INTERFACE I_Axis

METHOD PrepareDecoupling : I_Axis
VAR_INPUT
	slaveAxis : REFERENCE TO AXIS_REF;
	slaveStatus : REFERENCE TO ST_AXISSTATUS;
END_VAR
END_METHOD

METHOD StartCoupling : I_Axis
VAR_INPUT
END_VAR
END_METHOD

METHOD StartDecoupling : BOOL
VAR_INPUT
END_VAR
END_METHOD

METHOD StartHoming : BOOL;
VAR_INPUT
END_VAR
END_METHOD

END_INTERFACE

(* stored: Version 1.1.0.1, ProductVersion 3.1.4024.2
   Itf I_Axis: Id {e29f8469-a3e8-4cfa-a5ee-f4f6afb467e5}
   Method PrepareDecoupling: Id {54e06715-75df-426c-bd82-274c8cc90fa9}
   Method StartCoupling: Id {2c151b5b-bdad-4017-b369-02a28ecd6e66}
   Method StartDecoupling: Id {06b60ea2-3f04-453a-b850-2a578a6457e0}
   Method StartHoming: Id {365249dc-02da-41e0-bb2e-19d5dd02905e} *)
